// TwinCAT 3 PLC project PLC1
// ProgramVersion: 3.1.4024.0
// libraries:
//   Tc2_Standard, * (Beckhoff Automation GmbH)
//   Tc2_System, * (Beckhoff Automation GmbH)
//   Tc3_Module, * (Beckhoff Automation GmbH)
// project tree:
//   / PlcTask.TcTTO
//   SimpleFilter/ fnSimpleFilter.TcPOU, MAIN.TcPOU
// real-time tasks:
//   TASK PlcTask: cycle T#10ms, priority 20, ADS port 350

CONFIGURATION PLC1
    RESOURCE PLC ON TwinCAT3
        TASK PlcTask(INTERVAL := T#10ms, PRIORITY := 20);
        PROGRAM MAIN WITH PlcTask : MAIN;
    END_RESOURCE
END_CONFIGURATION

// ---- SimpleFilter/MAIN.TcPOU
PROGRAM MAIN
VAR
	rawValue		:REAL := 100;		// This can be a sensor
	
	rFilterSize		:REAL := 0.99;
	rFilteredValue	:REAL;
	bError 			:BOOL;
END_VAR

bError := fnSimpleFilter(UnfilterdValue := rawValue, FilterSize := rFilterSize, FilteredValue := rFilteredValue);

END_PROGRAM

// ---- SimpleFilter/fnSimpleFilter.TcPOU
FUNCTION fnSimpleFilter	: BOOL
VAR_INPUT
	UnfilterdValue	:REAL;					// Unfiltered (raw) value
	FilterSize		:REAL;					// Filter value (0.0 = No filter ; 1.0 = MAX. filter)
	FilteredValue	:REFERENCE TO REAL;		// Filtered value
END_VAR

(*
	FiltererValue = ( K * FiltererValue ) + ( (1-K) * NewValue )

	"Filter" must BE in range from 0 TO 1
	- 0.0: No filter
	- 0.5: Simular to average
	- 1.0: Strongest filter
*)
IF FilterSize <= 1.0
AND FilterSize >= 0.0
THEN
	// Filter sensor value
	FilteredValue := (FilterSize * FilteredValue) + ( (1.0 - FilterSize) * UnfilterdValue);
	fnSimpleFilter := TRUE;
ELSE
	fnSimpleFilter := FALSE;
END_IF

END_FUNCTION
